(* IEC 61131-3 sources: uPC2_EMCTEST/UPC2_EMCTEST/UPC2_EMCTEST/Source/Programs (part 2) *)

(* ---- 090_OutputMng.st ---- *)
USING System;
USING System.IO;

VAR_GLOBAL PERSISTENT
    (**Dout1 relè logic (FALSE=NO, TRUE=NC)*)
    Dout1Logic : BOOL := DOUT_LOGIC_NO;
END_VAR

PROGRAM OutputMng
    VAR PUBLIC
        (**Analog output 1 status*) {METADATA MIN_VAL 0.0} {METADATA MAX_VAL 100.0} {ATTRIBUTE UOM PERCENT}
        AOut1       : REAL;
    END_VAR

    {REGION DOut1}
        noConfig[1].enable    := TRUE;
        noConfig[1].mode_type := LIB_IO_STANDARD_RELE;
        //NO[1]                 := GblAlarm XOR Dout1Logic;
    {ENDREGION}

    {REGION AOut1}
        yConfig[1].mode_type := LIB_IO_OUT_0_10V;
        //Y[1]                 := TO_UINT(AOut1 * 10.0);
    {ENDREGION}
END_PROGRAM

(* ---- 900_NetFieldbus_Write.st ---- *)
USING System.Math;

PROGRAM NetFieldbus_Write

	IF En_FB1 THEN
    {REGION COMUNICATION BETWEEN CLIENT/SALVE BAORD}

        {REGION WRITES PARAMETERS INSIDE SERVER BOARD (COIL STATUS)}

            //..........................................
            // PUT HERE YOUR VARIABLEs
            //..........................................
//            ClientModbus_pCO.CS_0_UnitOn := UnitOn;
        {ENDREGION}

        {REGION WRITES PARAMETERS INSIDE SERVER BOARD (HOLDING REGISTERS)}

            //..........................................
            // PUT HERE YOUR VARIABLEs
            //..........................................

        {ENDREGION}
    {ENDREGION}
END_IF;

END_PROGRAM
